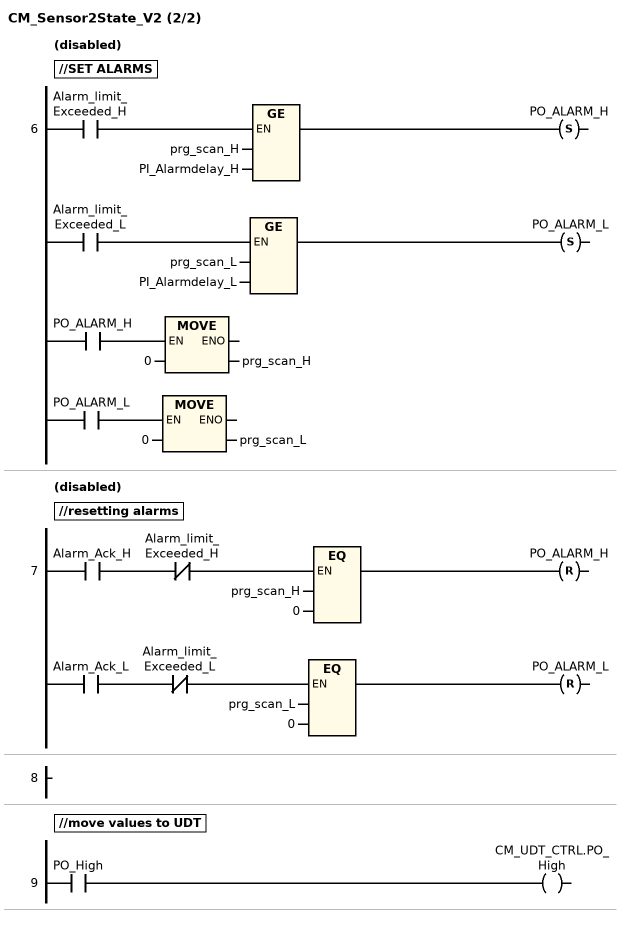
// NETWORK 6 (disabled)
// label: //SET ALARMS
// PO_ALARM_H S= Alarm_limit_Exceeded_H AND prg_scan_H >= PI_Alarmdelay_H;
// PO_ALARM_L S= Alarm_limit_Exceeded_L AND prg_scan_L >= PI_Alarmdelay_L;
// IF PO_ALARM_H THEN prg_scan_H := 0; END_IF
// IF PO_ALARM_L THEN prg_scan_L := 0; END_IF

// NETWORK 7 (disabled)
// label: //resetting alarms
// PO_ALARM_H R= Alarm_Ack_H AND NOT Alarm_limit_Exceeded_H AND prg_scan_H = 0;
// PO_ALARM_L R= Alarm_Ack_L AND NOT Alarm_limit_Exceeded_L AND prg_scan_L = 0;

// NETWORK 8

// NETWORK 9
// label: //move values to UDT
CM_UDT_CTRL.PO_High := PO_High;

END_FUNCTION_BLOCK

// ---- POUs/CM_V2/CM_SensorAnalog_V2.TcPOU
FUNCTION_BLOCK CM_SensorAnalog_V2
VAR_INPUT
	
	PI_ManualMode : BOOL;
	PI_AutoMode : BOOL;
	
	//ALARMS:
	PI_AlarmHighHighEnable : BOOL;
	PI_AlarmHighEnable : BOOL;
	PI_AlarmLowEnable : BOOL;
	PI_AlarmLowLowEnable : BOOL;
	
	PI_AlarmHighHighLimit : REAL;
	PI_AlarmHighLimit : REAL;
	PI_AlarmLowLimit : REAL;
	PI_AlarmLowLowLimit : REAL;
	
	PI_AlarmDelay_HH : LREAL;
	PI_AlarmDelay_H : LREAL;
	PI_AlarmDelay_L : LREAL;
	PI_AlarmDelay_LL : LREAL;
	
	PI_PV :DINT;
	
	
	ENABLE_SCALING : BOOL;
	PI_PV_MAX_IN : INT;
	PI_PV_MIN_IN : INT;
	PI_PV_MAX_OUT : INT;
	PI_PV_MIN_OUT : INT;
END_VAR
VAR_OUTPUT
	
	PO_PV_SCALED : REAL;

	PO_ALARM_HH : BOOL;
	PO_ALARM_H : BOOL;
	PO_ALARM_L : BOOL;
	PO_ALARM_LL : BOOL;
END_VAR
VAR
	scale : Tc2_ControllerToolbox.FB_CTRL_SCALE;
	scaleParams : ST_CTRL_SCALE_PARAMS;
	
	Alarm_limit_Exceeded_HH : BOOL;
	Alarm_limit_Exceeded_H : BOOL;
	Alarm_limit_Exceeded_L : BOOL;
	Alarm_limit_Exceeded_LL : BOOL;
	
	Alarm_Ack_HH : BOOL;
	Alarm_Ack_H : BOOL;
	Alarm_Ack_L : BOOL;
	Alarm_Ack_LL : BOOL;
	
	alarmDelay_HH : systemTimeDelay;
	alarmDelay_H : systemTimeDelay;
	alarmDelay_L : systemTimeDelay;
	alarmDelay_LL : systemTimeDelay;
	
	DelayForHistorianBit_HH: TON;
	DelayForHistorianBit_H: TON;
	DelayForHistorianBit_L: TON;
	DelayForHistorianBit_LL: TON;
	
	HIST_BIT_HH : BOOL;
	HIST_BIT_H : BOOL;
	HIST_BIT_L : BOOL;
	HIST_BIT_LL : BOOL;
END_VAR
VAR_IN_OUT
END_VAR

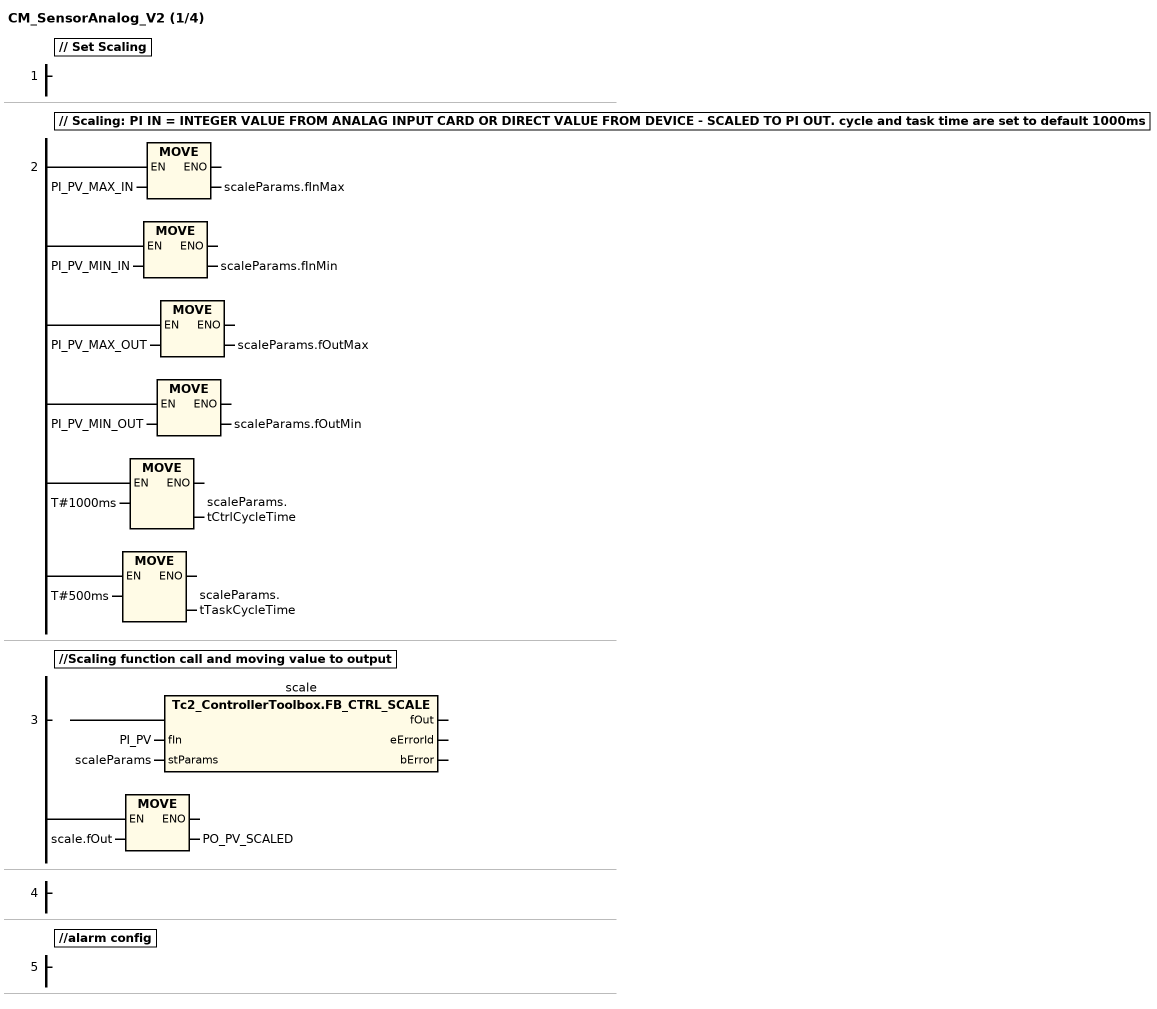
// NETWORK 1
// label: // Set Scaling

// NETWORK 2
// label: // Scaling: PI IN = INTEGER VALUE FROM ANALAG INPUT CARD OR DIRECT VALUE FROM DEVICE - SCALED TO PI OUT. cycle and task time are set to default 1000ms
scaleParams.fInMax := PI_PV_MAX_IN;
scaleParams.fInMin := PI_PV_MIN_IN;
scaleParams.fOutMax := PI_PV_MAX_OUT;
scaleParams.fOutMin := PI_PV_MIN_OUT;
scaleParams.tCtrlCycleTime := T#1000ms;
scaleParams.tTaskCycleTime := T#500ms;

// NETWORK 3
// label: //Scaling function call and moving value to output
scale(fIn := PI_PV, stParams := scaleParams); // Tc2_ControllerToolbox.FB_CTRL_SCALE
PO_PV_SCALED := scale.fOut;

// NETWORK 4

// NETWORK 5
// label: //alarm config

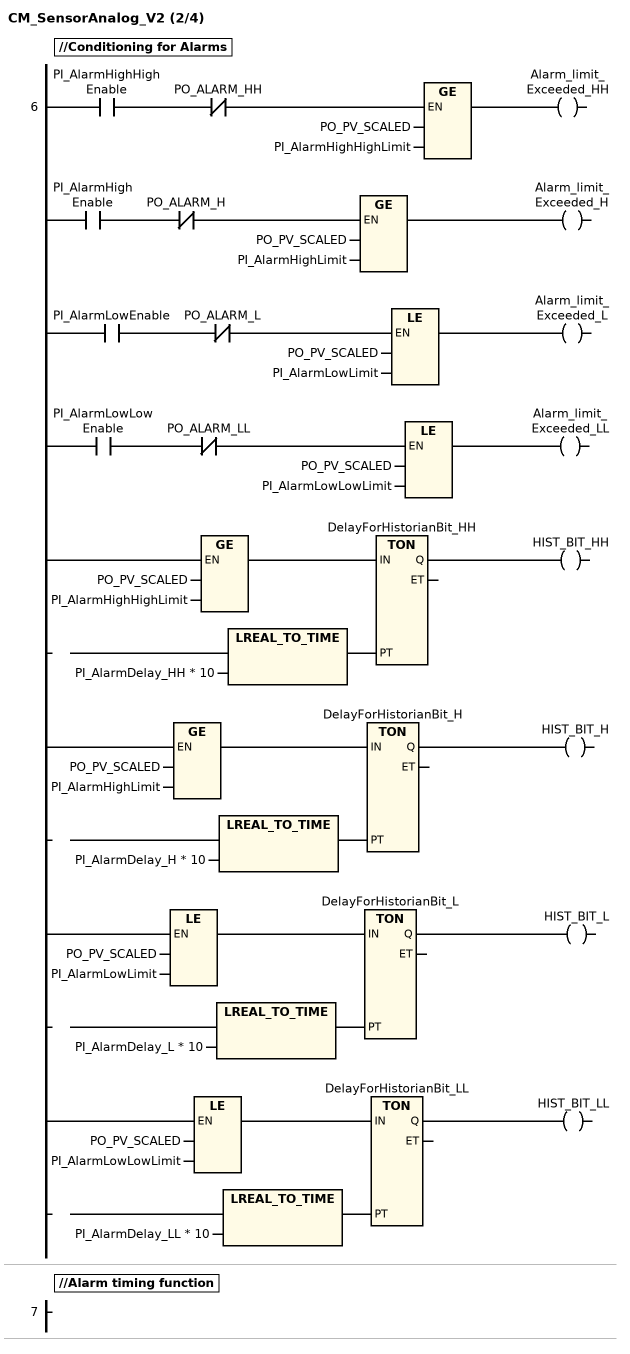
// NETWORK 6
// label: //Conditioning for Alarms
Alarm_limit_Exceeded_HH := PI_AlarmHighHighEnable AND NOT PO_ALARM_HH AND PO_PV_SCALED >= PI_AlarmHighHighLimit;
Alarm_limit_Exceeded_H := PI_AlarmHighEnable AND NOT PO_ALARM_H AND PO_PV_SCALED >= PI_AlarmHighLimit;
Alarm_limit_Exceeded_L := PI_AlarmLowEnable AND NOT PO_ALARM_L AND PO_PV_SCALED <= PI_AlarmLowLimit;
Alarm_limit_Exceeded_LL := PI_AlarmLowLowEnable AND NOT PO_ALARM_LL AND PO_PV_SCALED <= PI_AlarmLowLowLimit;
DelayForHistorianBit_HH(IN := PO_PV_SCALED >= PI_AlarmHighHighLimit, PT := LREAL_TO_TIME(PI_AlarmDelay_HH * 10)); // TON
HIST_BIT_HH := DelayForHistorianBit_HH.Q;
DelayForHistorianBit_H(IN := PO_PV_SCALED >= PI_AlarmHighLimit, PT := LREAL_TO_TIME(PI_AlarmDelay_H * 10)); // TON
HIST_BIT_H := DelayForHistorianBit_H.Q;
DelayForHistorianBit_L(IN := PO_PV_SCALED <= PI_AlarmLowLimit, PT := LREAL_TO_TIME(PI_AlarmDelay_L * 10)); // TON
HIST_BIT_L := DelayForHistorianBit_L.Q;
DelayForHistorianBit_LL(IN := PO_PV_SCALED <= PI_AlarmLowLowLimit, PT := LREAL_TO_TIME(PI_AlarmDelay_LL * 10)); // TON
HIST_BIT_LL := DelayForHistorianBit_LL.Q;

// NETWORK 7
// label: //Alarm timing function

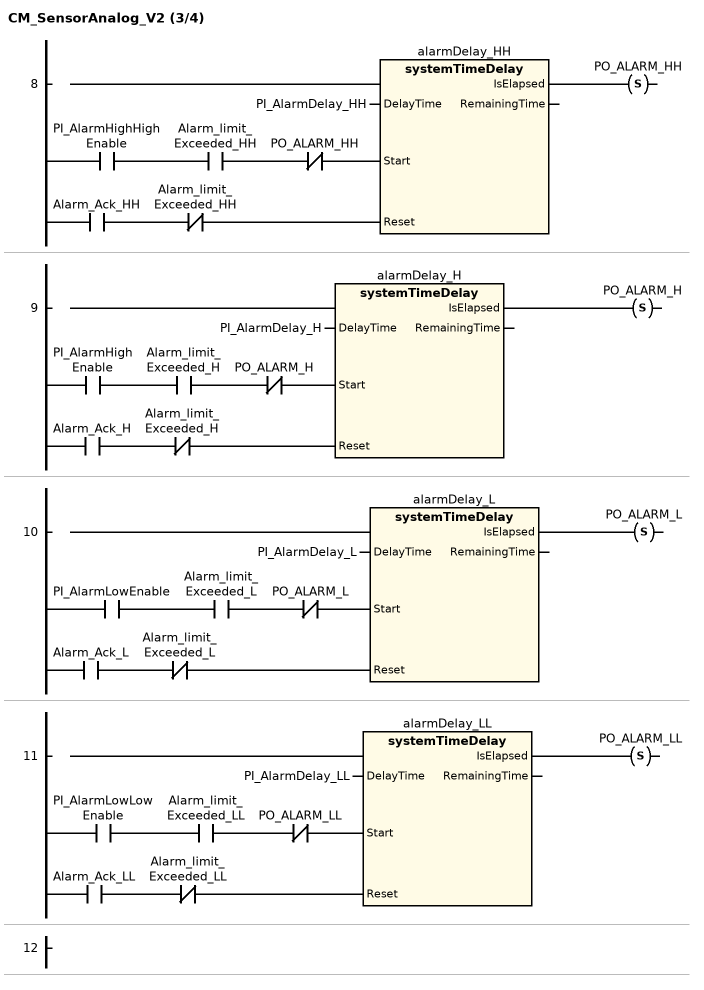
// NETWORK 8
alarmDelay_HH(
    DelayTime := PI_AlarmDelay_HH,
    Start := PI_AlarmHighHighEnable AND Alarm_limit_Exceeded_HH AND NOT PO_ALARM_HH,
    Reset := Alarm_Ack_HH AND NOT Alarm_limit_Exceeded_HH); // systemTimeDelay
PO_ALARM_HH S= alarmDelay_HH.IsElapsed;

// NETWORK 9
alarmDelay_H(
    DelayTime := PI_AlarmDelay_H,
    Start := PI_AlarmHighEnable AND Alarm_limit_Exceeded_H AND NOT PO_ALARM_H,
    Reset := Alarm_Ack_H AND NOT Alarm_limit_Exceeded_H); // systemTimeDelay
PO_ALARM_H S= alarmDelay_H.IsElapsed;

// NETWORK 10
alarmDelay_L(
    DelayTime := PI_AlarmDelay_L,
    Start := PI_AlarmLowEnable AND Alarm_limit_Exceeded_L AND NOT PO_ALARM_L,
    Reset := Alarm_Ack_L AND NOT Alarm_limit_Exceeded_L); // systemTimeDelay
PO_ALARM_L S= alarmDelay_L.IsElapsed;

// NETWORK 11
alarmDelay_LL(
    DelayTime := PI_AlarmDelay_LL,
    Start := PI_AlarmLowLowEnable AND Alarm_limit_Exceeded_LL AND NOT PO_ALARM_LL,
    Reset := Alarm_Ack_LL AND NOT Alarm_limit_Exceeded_LL); // systemTimeDelay
PO_ALARM_LL S= alarmDelay_LL.IsElapsed;

// NETWORK 12

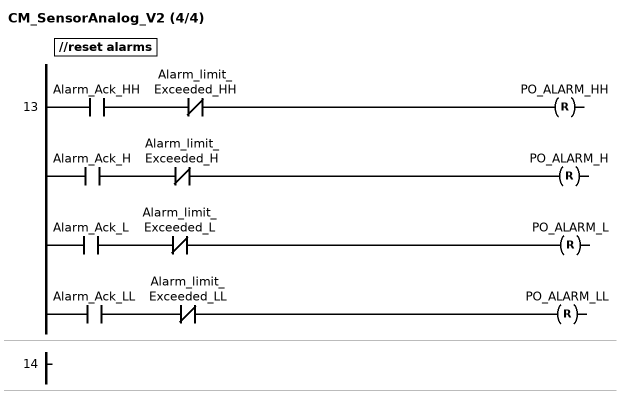
// NETWORK 13
// label: //reset alarms
PO_ALARM_HH R= Alarm_Ack_HH AND NOT Alarm_limit_Exceeded_HH;
PO_ALARM_H R= Alarm_Ack_H AND NOT Alarm_limit_Exceeded_H;
PO_ALARM_L R= Alarm_Ack_L AND NOT Alarm_limit_Exceeded_L;
PO_ALARM_LL R= Alarm_Ack_LL AND NOT Alarm_limit_Exceeded_LL;

// NETWORK 14

END_FUNCTION_BLOCK

// ---- POUs/Control functions/FB_PID.TcPOU
FUNCTION_BLOCK FB_PID
VAR_INPUT
	Manual_mode : BOOL;
	Auto_mode : BOOL;
	
	fSetpointValue					: LREAL;
	fActualValue					: LREAL;
	fManSyncValue					: LREAL;
	bSync							: BOOL;
	
	IN_stCTRL_PID_PARAMS				: ST_CTRL_PID_PARAMS;
END_VAR
VAR_OUTPUT
	fOut							: LREAL;
	bHold							: BOOL;
END_VAR
VAR
	eMode							: E_CTRL_MODE;
	stCTRL_PID_PARAMS				: ST_CTRL_PID_PARAMS;
	

	eErrorId						: E_CTRL_ERRORCODES;
	bError							: BOOL;
	bARWactive						: BOOL;
	
	(* controller *)
	fbCTRL_PID						: FB_CTRL_PID;

	bInit							: BOOL	:= TRUE;
	fbTON							: TON;
END_VAR

IF Manual_mode THEN
	eMode :=  4;
END_IF
IF Auto_mode THEN
	eMode :=  2;
ELSE
	eMode :=  0;	
END_IF

IF bInit THEN
	
	stCTRL_PID_PARAMS := IN_stCTRL_PID_PARAMS;
	(*
	(* init parameter struct *)
	stCTRL_PID_PARAMS.tCtrlCycleTime		:= T#500MS;	//used to control the actual sample time of the PID algorythm, must be = or > than the task cycle time
	stCTRL_PID_PARAMS.tTaskCycleTime		:= T#100MS;		// must be the same as the cycletime configured in the task which the regulator is called in (CyclicTask100Ms)
	stCTRL_PID_PARAMS.fKp					:= 5.0;			(* proportional gain Kp				*)
	stCTRL_PID_PARAMS.tTn					:= T#100S;		(*  Tn								*)
	stCTRL_PID_PARAMS.tTv					:= T#200MS;		(*  Tv								*)
	stCTRL_PID_PARAMS.tTd					:= T#500MS;		(*  Td								*)
	stCTRL_PID_PARAMS.fOutMaxLimit			:=  100.0;			(* maximum output limit			(for  fillValve)	*) 
	stCTRL_PID_PARAMS.fOutMinLimit			:= -0.0;			(* minimum output limit			(for  fillValve)	*)
	
	
	*)
	(* set the mode to ACTIVE --> normal operation *)
	
	eMode := eCTRL_MODE_ACTIVE;

	(* reset the init flag *)
	bInit := FALSE;
END_IF
IF bInit AND eMode = 4 THEN
	
	stCTRL_PID_PARAMS := IN_stCTRL_PID_PARAMS;
	(* init parameter struct *)

	(* set the mode to ACTIVE --> normal operation *)
	eMode := eCTRL_MODE_ACTIVE;

	(* reset the init flag *)
	bInit := FALSE;
END_IF

(* call controller *)
fbCTRL_PID(		fSetpointValue		:= fSetpointValue,
				fActualValue		:= fActualValue, //feedback value (proces variable)
				fManSyncValue		:= fManSyncValue, // controll fOut directly with 0-100 %?
				bSync				:= bSync,
				eMode				:= eMode,
				bHold				:= bHold,
				stParams			:= stCTRL_PID_PARAMS,
				fOut				=> fOut, // output to PID
				bARWactive			=> bARWactive,
				eErrorId			=> eErrorId,
				bError				=> bError
				);

END_FUNCTION_BLOCK

// ---- POUs/EM/EM_Tank.TcPOU
FUNCTION_BLOCK EM_Tank
VAR_INPUT
	
END_VAR
VAR_OUTPUT
END_VAR
VAR
END_VAR

END_FUNCTION_BLOCK

// ---- POUs/Plant Control/FB_PlantControl.TcPOU
FUNCTION_BLOCK FB_PlantControl
VAR_INPUT
	
	PI_on : BOOL;
	
	PI_Auto : BOOL;
	PI_Manual : BOOL;
	
	PI_Start : BOOL;
	PI_Stop : BOOL;
	PI_Reset : BOOL;
	PI_EmgStop : BOOL;
	
END_VAR
VAR_OUTPUT
	PO_ON : BOOL;
	
	PO_Auto : BOOL;
	PO_Manual : BOOL;
	
	PO_Startet : BOOL;
	PO_Stopped : BOOL;
	PO_Reset : BOOL;
	PO_ResetEmgStop_5s :BOOL;
	
	PO_EmgStopped : BOOL;
	
	PO_Mode_Control : ENUM_MODE_HANDLER;
	
END_VAR
VAR
	EmgResetTimerOff : Tc2_Standard.TON;
	
END_VAR
VAR_IN_OUT
	
	SCADA_Ctrl_Plant : Udt_PlantControl;
	
END_VAR

VAR CONSTANT
	SR_Auto: SR;
	SR_Man : SR;
	
	SR_start : SR;
	SR_Stop : SR;
	SR_EMGStop: SR;
	
END_VAR

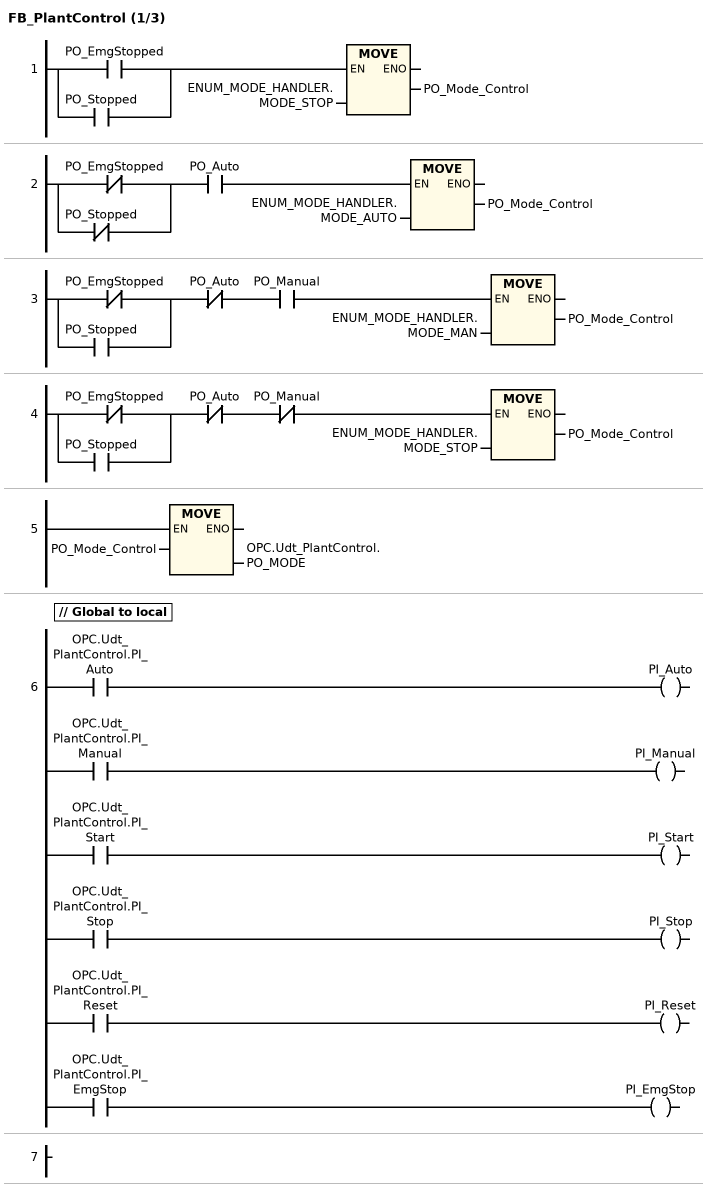
// NETWORK 1
IF PO_EmgStopped OR PO_Stopped THEN PO_Mode_Control := ENUM_MODE_HANDLER.MODE_STOP; END_IF

// NETWORK 2
IF (NOT PO_EmgStopped OR NOT PO_Stopped) AND PO_Auto THEN PO_Mode_Control := ENUM_MODE_HANDLER.MODE_AUTO; END_IF

// NETWORK 3
IF (NOT PO_EmgStopped OR PO_Stopped) AND NOT PO_Auto AND PO_Manual THEN
    PO_Mode_Control := ENUM_MODE_HANDLER.MODE_MAN;
END_IF

// NETWORK 4
IF (NOT PO_EmgStopped OR PO_Stopped) AND NOT PO_Auto AND NOT PO_Manual THEN
    PO_Mode_Control := ENUM_MODE_HANDLER.MODE_STOP;
END_IF

// NETWORK 5
OPC.Udt_PlantControl.PO_MODE := PO_Mode_Control;

// NETWORK 6
// label: // Global to local
PI_Auto := OPC.Udt_PlantControl.PI_Auto;
PI_Manual := OPC.Udt_PlantControl.PI_Manual;
PI_Start := OPC.Udt_PlantControl.PI_Start;
PI_Stop := OPC.Udt_PlantControl.PI_Stop;
PI_Reset := OPC.Udt_PlantControl.PI_Reset;
PI_EmgStop := OPC.Udt_PlantControl.PI_EmgStop;

// NETWORK 7

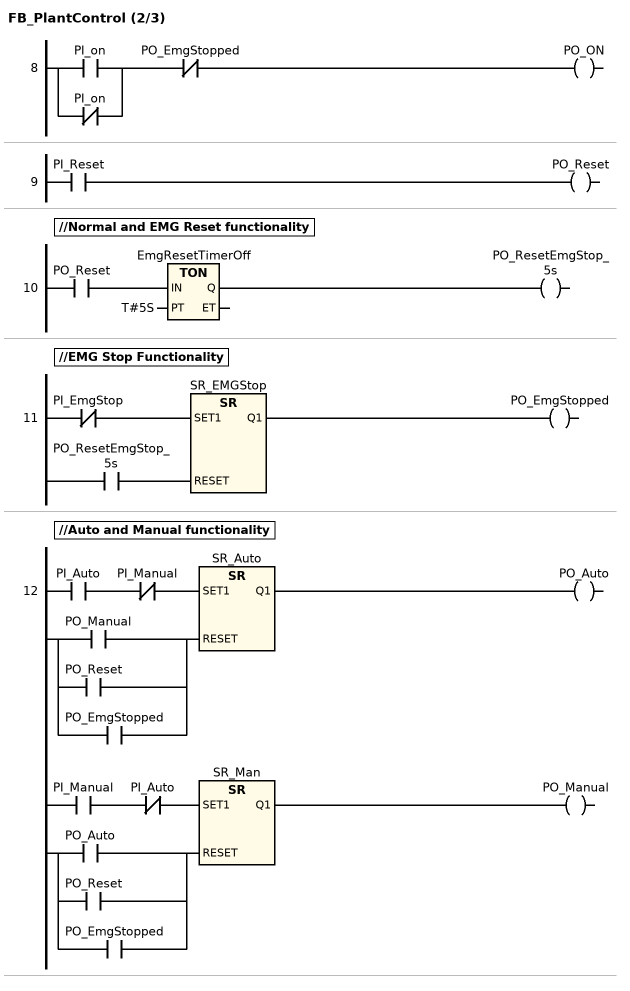
// NETWORK 8
PO_ON := (PI_on OR NOT PI_on) AND NOT PO_EmgStopped;

// NETWORK 9
PO_Reset := PI_Reset;

// NETWORK 10
// label: //Normal and EMG Reset functionality
EmgResetTimerOff(IN := PO_Reset, PT := T#5S); // TON
PO_ResetEmgStop_5s := EmgResetTimerOff.Q;

// NETWORK 11
// label: //EMG Stop Functionality
SR_EMGStop(SET1 := NOT PI_EmgStop, RESET := PO_ResetEmgStop_5s); // SR
PO_EmgStopped := SR_EMGStop.Q1;

// NETWORK 12
// label: //Auto and Manual functionality
SR_Auto(SET1 := PI_Auto AND NOT PI_Manual, RESET := PO_Manual OR PO_Reset OR PO_EmgStopped); // SR
PO_Auto := SR_Auto.Q1;
SR_Man(SET1 := PI_Manual AND NOT PI_Auto, RESET := PO_Auto OR PO_Reset OR PO_EmgStopped); // SR
PO_Manual := SR_Man.Q1;

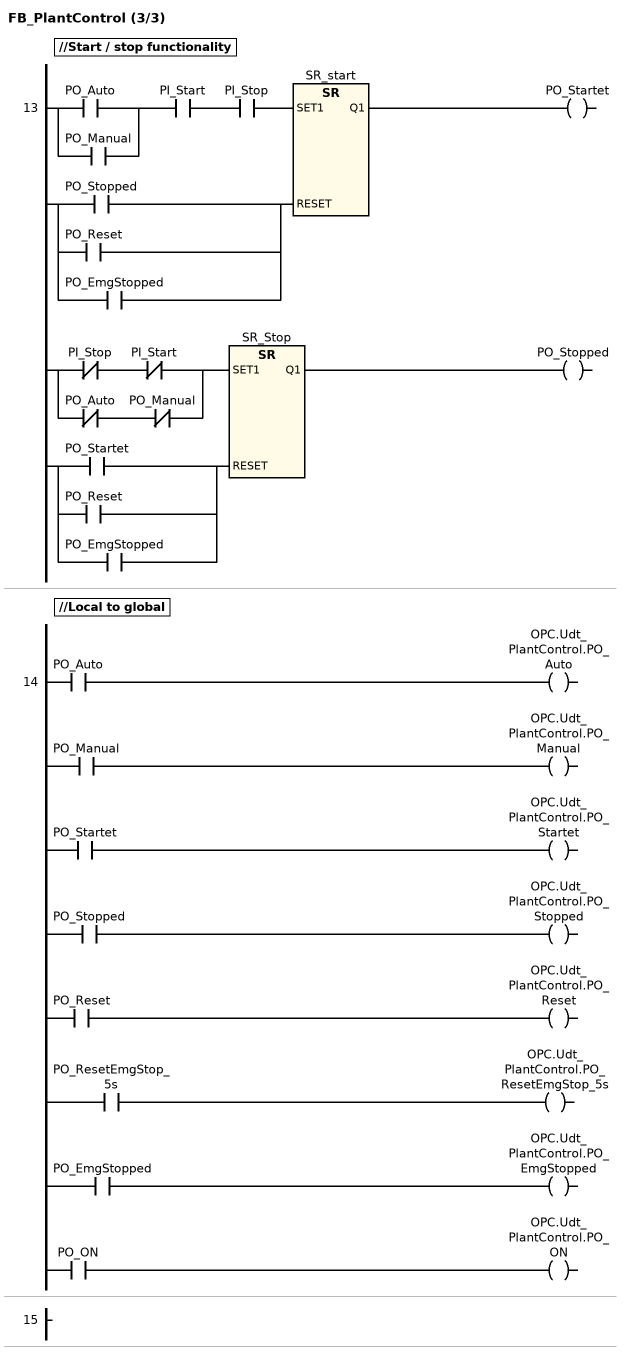
// NETWORK 13
// label: //Start / stop functionality
SR_start(SET1 := (PO_Auto OR PO_Manual) AND PI_Start AND PI_Stop, RESET := PO_Stopped OR PO_Reset OR PO_EmgStopped); // SR
PO_Startet := SR_start.Q1;
SR_Stop(SET1 := NOT PI_Stop AND NOT PI_Start OR NOT PO_Auto AND NOT PO_Manual, RESET := PO_Startet OR PO_Reset OR PO_EmgStopped); // SR
PO_Stopped := SR_Stop.Q1;

// NETWORK 14
// label: //Local to global
OPC.Udt_PlantControl.PO_Auto := PO_Auto;
OPC.Udt_PlantControl.PO_Manual := PO_Manual;
OPC.Udt_PlantControl.PO_Startet := PO_Startet;
OPC.Udt_PlantControl.PO_Stopped := PO_Stopped;
OPC.Udt_PlantControl.PO_Reset := PO_Reset;
OPC.Udt_PlantControl.PO_ResetEmgStop_5s := PO_ResetEmgStop_5s;
OPC.Udt_PlantControl.PO_EmgStopped := PO_EmgStopped;
OPC.Udt_PlantControl.PO_ON := PO_ON;

// NETWORK 15

END_FUNCTION_BLOCK

// ---- POUs/Plant Control/FB_PlantControl_V2.TcPOU
FUNCTION_BLOCK FB_PlantControl_V2
VAR_INPUT
	Plant_ID : STRING;
	
	PI_on : BOOL;
	
	PI_Auto : BOOL;
	PI_Manual : BOOL;
	
	PI_Start : BOOL;
	PI_Stop : BOOL;
	PI_Reset : BOOL;
	PI_EmgStop : BOOL;
	
END_VAR
VAR_OUTPUT
	PO_ON : BOOL;
	
	PO_Auto : BOOL;
	PO_Manual : BOOL;
	
	PO_Startet : BOOL;
	PO_Stopped : BOOL;
	PO_Reset : BOOL;
	PO_ResetEmgStop_5s :BOOL;
	
	PO_EmgStopped : BOOL;
	
	PO_Mode_Control : ENUM_MODE_HANDLER;
	
END_VAR
VAR
	EmgResetTimerOff : Tc2_Standard.TON;
	
END_VAR
VAR_IN_OUT
END_VAR

VAR CONSTANT
	SR_Auto: SR;
	SR_Man : SR;
	
	SR_start : SR;
	SR_Stop : SR;
	SR_EMGStop: SR;
	
END_VAR

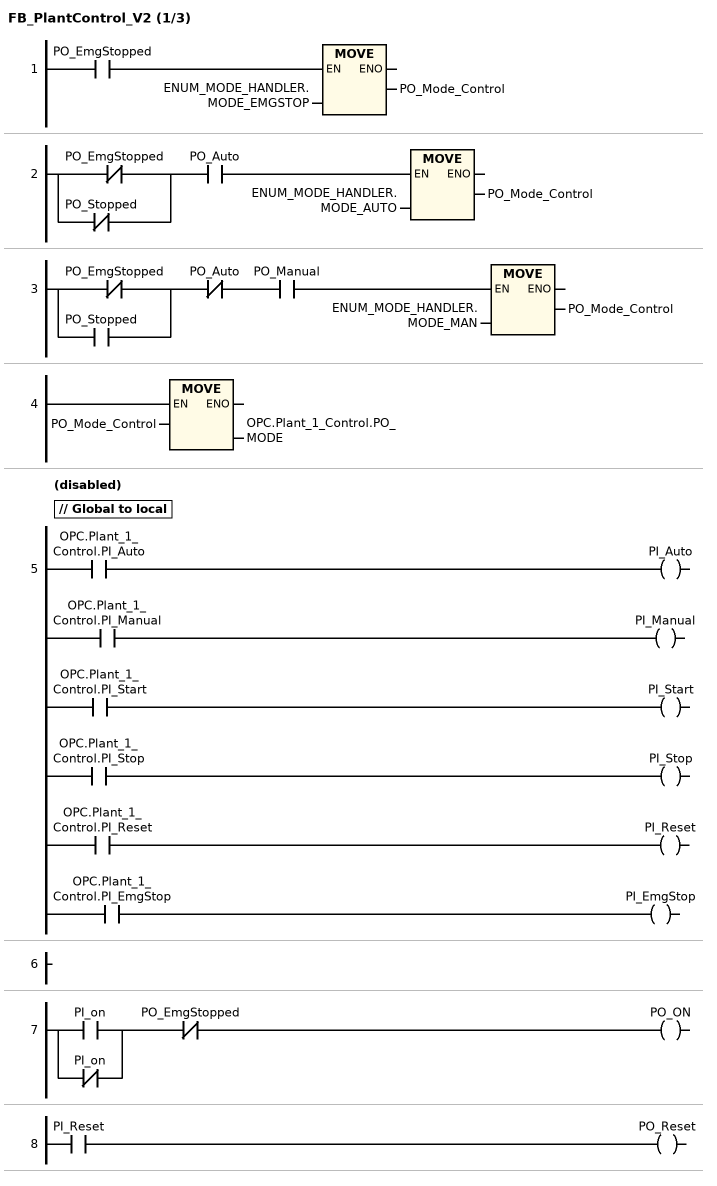
// NETWORK 1
IF PO_EmgStopped THEN PO_Mode_Control := ENUM_MODE_HANDLER.MODE_EMGSTOP; END_IF

// NETWORK 2
IF (NOT PO_EmgStopped OR NOT PO_Stopped) AND PO_Auto THEN PO_Mode_Control := ENUM_MODE_HANDLER.MODE_AUTO; END_IF

// NETWORK 3
IF (NOT PO_EmgStopped OR PO_Stopped) AND NOT PO_Auto AND PO_Manual THEN
    PO_Mode_Control := ENUM_MODE_HANDLER.MODE_MAN;
END_IF

// NETWORK 4
OPC.Plant_1_Control.PO_MODE := PO_Mode_Control;

// NETWORK 5 (disabled)
// label: // Global to local
// PI_Auto := OPC.Plant_1_Control.PI_Auto;
// PI_Manual := OPC.Plant_1_Control.PI_Manual;
// PI_Start := OPC.Plant_1_Control.PI_Start;
// PI_Stop := OPC.Plant_1_Control.PI_Stop;
// PI_Reset := OPC.Plant_1_Control.PI_Reset;
// PI_EmgStop := OPC.Plant_1_Control.PI_EmgStop;

// NETWORK 6

// NETWORK 7
PO_ON := (PI_on OR NOT PI_on) AND NOT PO_EmgStopped;

// NETWORK 8
PO_Reset := PI_Reset;

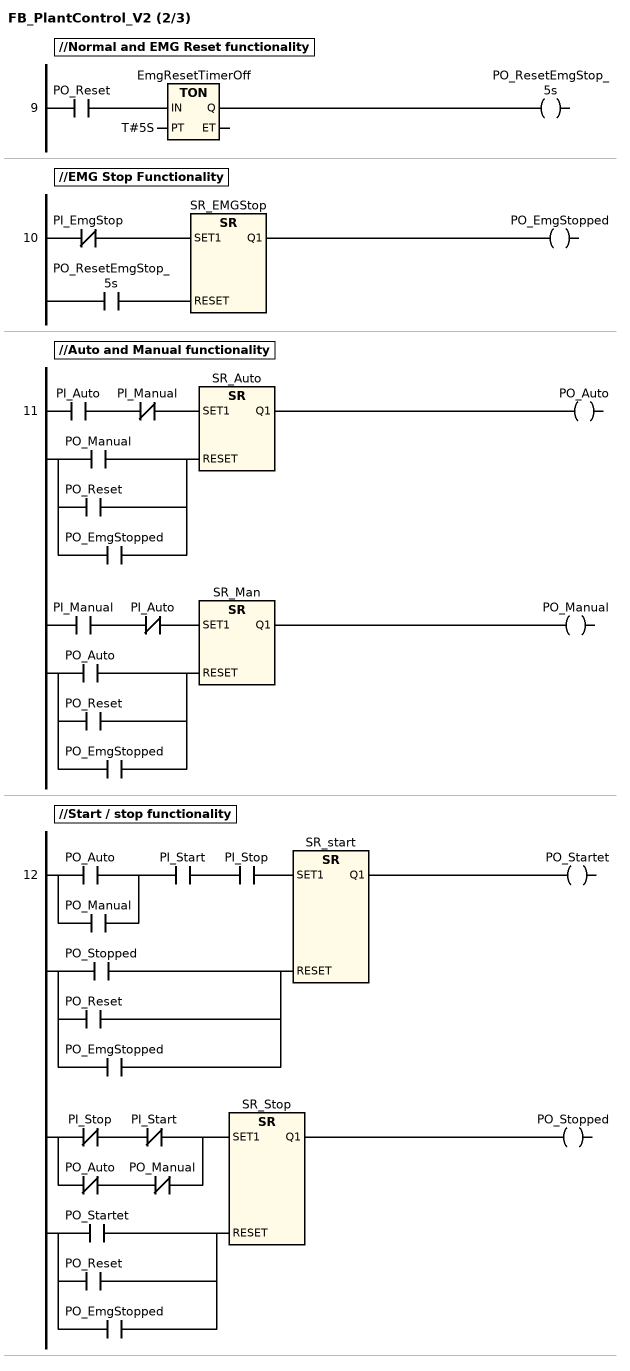
// NETWORK 9
// label: //Normal and EMG Reset functionality
EmgResetTimerOff(IN := PO_Reset, PT := T#5S); // TON
PO_ResetEmgStop_5s := EmgResetTimerOff.Q;

// NETWORK 10
// label: //EMG Stop Functionality
SR_EMGStop(SET1 := NOT PI_EmgStop, RESET := PO_ResetEmgStop_5s); // SR
PO_EmgStopped := SR_EMGStop.Q1;

// NETWORK 11
// label: //Auto and Manual functionality
SR_Auto(SET1 := PI_Auto AND NOT PI_Manual, RESET := PO_Manual OR PO_Reset OR PO_EmgStopped); // SR
PO_Auto := SR_Auto.Q1;
SR_Man(SET1 := PI_Manual AND NOT PI_Auto, RESET := PO_Auto OR PO_Reset OR PO_EmgStopped); // SR
PO_Manual := SR_Man.Q1;

// NETWORK 12
// label: //Start / stop functionality
SR_start(SET1 := (PO_Auto OR PO_Manual) AND PI_Start AND PI_Stop, RESET := PO_Stopped OR PO_Reset OR PO_EmgStopped); // SR
PO_Startet := SR_start.Q1;
SR_Stop(SET1 := NOT PI_Stop AND NOT PI_Start OR NOT PO_Auto AND NOT PO_Manual, RESET := PO_Startet OR PO_Reset OR PO_EmgStopped); // SR
PO_Stopped := SR_Stop.Q1;

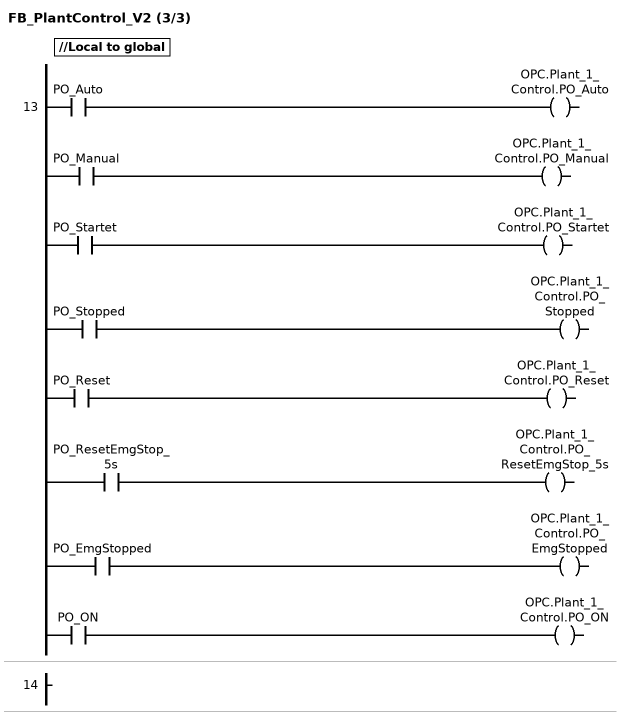
// NETWORK 13
// label: //Local to global
OPC.Plant_1_Control.PO_Auto := PO_Auto;
OPC.Plant_1_Control.PO_Manual := PO_Manual;
OPC.Plant_1_Control.PO_Startet := PO_Startet;
OPC.Plant_1_Control.PO_Stopped := PO_Stopped;
OPC.Plant_1_Control.PO_Reset := PO_Reset;
OPC.Plant_1_Control.PO_ResetEmgStop_5s := PO_ResetEmgStop_5s;
OPC.Plant_1_Control.PO_EmgStopped := PO_EmgStopped;
OPC.Plant_1_Control.PO_ON := PO_ON;

// NETWORK 14

END_FUNCTION_BLOCK

// ---- POUs/Scaling/FB_ScaleIN_1.TcPOU
FUNCTION_BLOCK FB_ScaleIN_1
VAR_INPUT
	inputForScaling : REAL;
	inMin : REAL;
	inMax : REAL;
	outMin : REAL;
	outMax : REAL;
	ctrlCycletime : TIME;
	taskCycletime : TIME;
END_VAR
VAR_OUTPUT
	scaledOutputInt : DINT;
	scaledOutputReal : REAL;
END_VAR
VAR
	fbScale : FB_CTRL_SCALE;
	stParamsForScaling : ST_CTRL_SCALE_PARAMS;
	
END_VAR

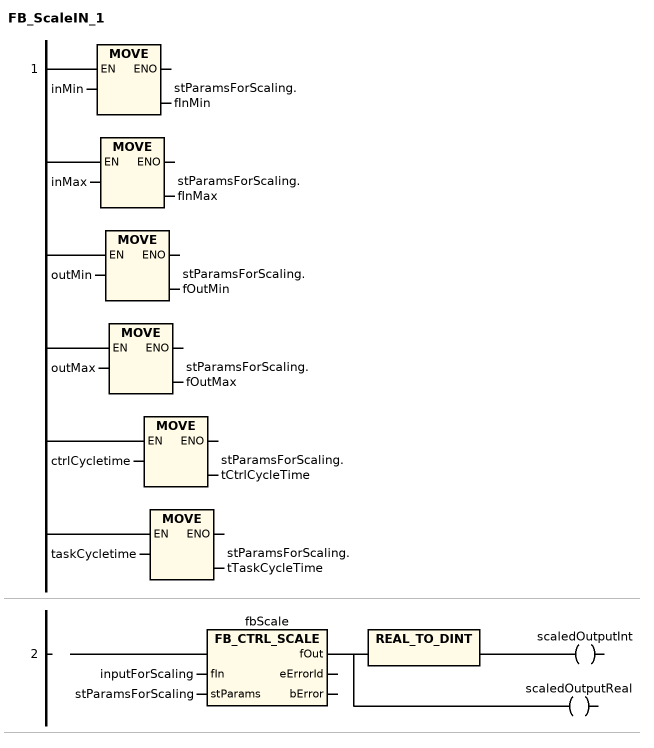
// NETWORK 1
stParamsForScaling.fInMin := inMin;
stParamsForScaling.fInMax := inMax;
stParamsForScaling.fOutMin := outMin;
stParamsForScaling.fOutMax := outMax;
stParamsForScaling.tCtrlCycleTime := ctrlCycletime;
stParamsForScaling.tTaskCycleTime := taskCycletime;

// NETWORK 2
fbScale(fIn := inputForScaling, stParams := stParamsForScaling); // FB_CTRL_SCALE
scaledOutputInt := REAL_TO_DINT(fbScale.fOut);
scaledOutputReal := fbScale.fOut;

END_FUNCTION_BLOCK

// ---- POUs/Scaling/FB_ScaleOut_1.TcPOU
FUNCTION_BLOCK FB_ScaleOut_1
VAR_INPUT
	inputForScaling : REAL;
	inMin : REAL;
	inMax : REAL;
	outMin : REAL;
	outMax : REAL;
	ctrlCycletime : TIME;
	taskCycletime : TIME;
END_VAR
VAR_OUTPUT
	scaledOutput : real;
END_VAR
VAR
	fbScale : FB_CTRL_SCALE;
	stParamsForScaling : ST_CTRL_SCALE_PARAMS;
	
END_VAR

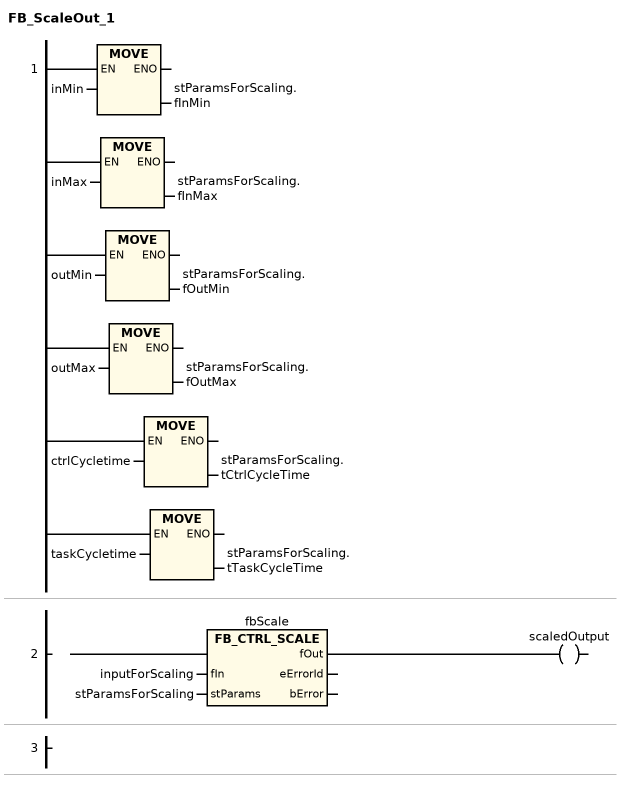
// NETWORK 1
stParamsForScaling.fInMin := inMin;
stParamsForScaling.fInMax := inMax;
stParamsForScaling.fOutMin := outMin;
stParamsForScaling.fOutMax := outMax;
stParamsForScaling.tCtrlCycleTime := ctrlCycletime;
stParamsForScaling.tTaskCycleTime := taskCycletime;

// NETWORK 2
fbScale(fIn := inputForScaling, stParams := stParamsForScaling); // FB_CTRL_SCALE
scaledOutput := fbScale.fOut;

// NETWORK 3

END_FUNCTION_BLOCK

// ---- POUs/System/FB_ScaleIN.TcPOU
FUNCTION_BLOCK FB_ScaleIN
VAR_INPUT
	inputForScaling : REAL;
	inMin : REAL;
	inMax : REAL;
	outMin : REAL;
	outMax : REAL;
	ctrlCycletime : TIME;
	taskCycletime : TIME;
END_VAR
VAR_OUTPUT
	scaledOutputInt : DINT;
	scaledOutputReal : REAL;
END_VAR
VAR
	fbScale : FB_CTRL_SCALE;
	stParamsForScaling : ST_CTRL_SCALE_PARAMS;
	
END_VAR

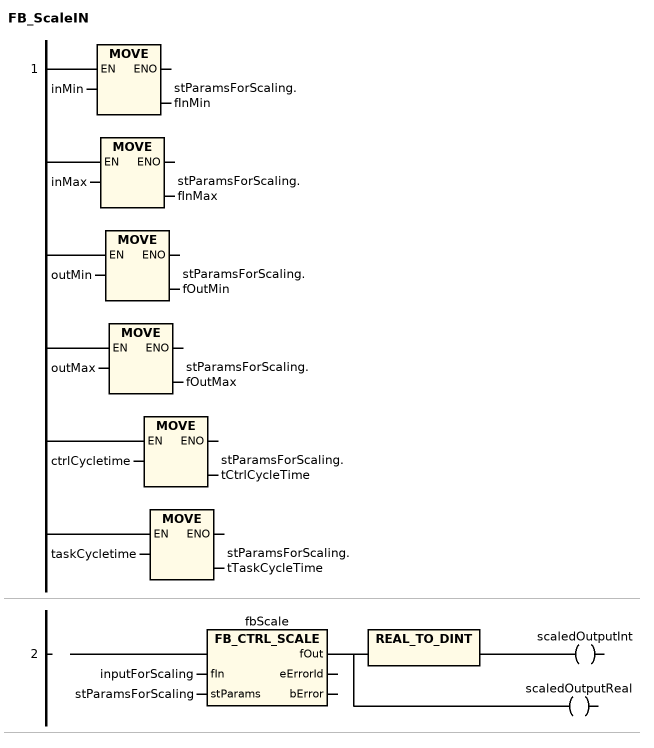
// NETWORK 1
stParamsForScaling.fInMin := inMin;
stParamsForScaling.fInMax := inMax;
stParamsForScaling.fOutMin := outMin;
stParamsForScaling.fOutMax := outMax;
stParamsForScaling.tCtrlCycleTime := ctrlCycletime;
stParamsForScaling.tTaskCycleTime := taskCycletime;

// NETWORK 2
fbScale(fIn := inputForScaling, stParams := stParamsForScaling); // FB_CTRL_SCALE
scaledOutputInt := REAL_TO_DINT(fbScale.fOut);
scaledOutputReal := fbScale.fOut;

END_FUNCTION_BLOCK

// ---- POUs/System/FB_ScaleOut.TcPOU
FUNCTION_BLOCK FB_ScaleOut
VAR_INPUT
	inputForScaling : REAL;
	inMin : REAL;
	inMax : REAL;
	outMin : REAL;
	outMax : REAL;
	ctrlCycletime : TIME;
	taskCycletime : TIME;
END_VAR
VAR_OUTPUT
	scaledOutput : real;
END_VAR
VAR
	fbScale : FB_CTRL_SCALE;
	stParamsForScaling : ST_CTRL_SCALE_PARAMS;
	
END_VAR

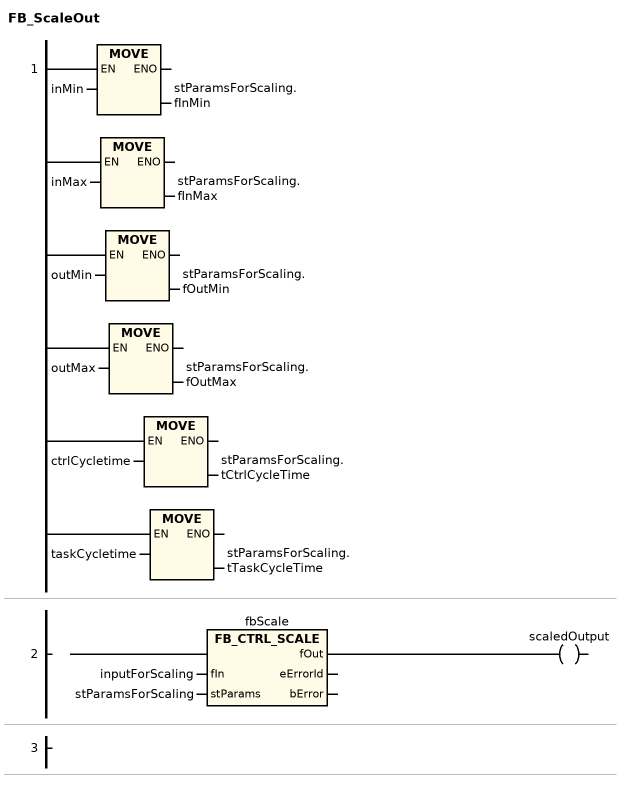
// NETWORK 1
stParamsForScaling.fInMin := inMin;
stParamsForScaling.fInMax := inMax;
stParamsForScaling.fOutMin := outMin;
stParamsForScaling.fOutMax := outMax;
stParamsForScaling.tCtrlCycleTime := ctrlCycletime;
stParamsForScaling.tTaskCycleTime := taskCycletime;

// NETWORK 2
fbScale(fIn := inputForScaling, stParams := stParamsForScaling); // FB_CTRL_SCALE
scaledOutput := fbScale.fOut;

// NETWORK 3

END_FUNCTION_BLOCK

// ---- POUs/System/SystemTimeTick.TcPOU
FUNCTION_BLOCK SystemTimeTick
VAR_INPUT
END_VAR
VAR_OUTPUT
END_VAR
VAR
	currentTicks : ULINT;
    timeMs : ULINT;
	timeS        : ULINT;  // seconds
    timeM        : ULINT;  // minutes
    timeH        : ULINT;  // hours
END_VAR

currentTicks := Tc2_System.F_GetSystemTime(); // returns system ticks

timeMs := currentTicks / 10000;   // convert to milliseconds (1 tick = 100ns)
timeS  := timeMs / 1000;                  // convert to seconds
timeM  := timeS / 60;                     // convert to minutes
timeH  := timeM / 60;                     // convert to hours

END_FUNCTION_BLOCK
